TYPE ST_PidParameters :
STRUCT
	Iterationtime: REAL;
	PB: REAL;
	Ti: REAL;
	Td: REAL;
	Bias: REAL;
END_STRUCT
END_TYPE

(* stored: Version 1.1.0.1, ProductVersion 3.1.4024.9
   DUT ST_PidParameters: Id {a5cba726-e634-473c-a420-6dfe234c8234} *)
